// TIA Portal project "MedicalTableS71500" (V15.1)

(* hardware
DEVICE "S71500/ET200MP-Station_1"  S7-1500 station
   slot 0: "Profilschiene_0"  Rack  6ES7 590-1***0-0AA0
   slot 1: "PLC_1"  CPU 1513-1 PN  6ES7 513-1AL02-0AB0  V2.6
      slot 3: "CPU-Display_1"  6ES7591-1AA00-0AA0
   slot 2: "DI 32x24VDC BA_1"  DI 32x24VDC BA  6ES7 521-1BL10-0AA0  V1.0
   slot 3: "AI 8xU/I/RTD/TC ST_1"  AI 8xU/I/RTD/TC ST  6ES7 531-7KF00-0AB0  V2.2
   slot 4: "DQ 32x24VDC/0.5A BA_1"  DQ 32x24VDC/0.5A BA  6ES7 522-1BL10-0AA0  V1.0
   slot 5: "AQ 4xU/I ST_1"  AQ 4xU/I ST  6ES7 532-5HD00-0AB0  V2.2
   slot 6: "DI 16x24VDC BA_1"  DI 16x24VDC BA  6ES7 521-1BH10-0AA0  V1.0
*)

// ===== PLC "PLC_1"  CPU 1513-1 PN =====

VAR_GLOBAL   // PLC tag table "Standard-Variablentabelle"
   "FlagControlOn" AT %M0.0 : Bool;
   "FlagM1ManualPosToMin" AT %M0.1 : Bool;
   "FlagM1ManualPosToMax" AT %M0.2 : Bool;
   "FlagM2ManualPosToMin" AT %M0.3 : Bool;
   "FlagM2ManualPosToMax" AT %M0.4 : Bool;
   "FlagM3ManualPosToMin" AT %M0.5 : Bool;
   "FlagM3ManualPosToMax" AT %M0.6 : Bool;
   "FlagM4ManualPosToMin" AT %M0.7 : Bool;
   "FlagM4ManualPosToMax" AT %M1.0 : Bool;
   "FlagEdgeHelperS5" AT %M1.1 : Bool;
   "FlagEdgeHelperS10" AT %M1.2 : Bool;
   "P2AllPositionsReached" AT %A2.2 : Bool;
   "P3M1PosReached" AT %A2.3 : Bool;
   "P4M2PosReached" AT %A2.4 : Bool;
   "P5M3PosReached" AT %A2.5 : Bool;
   "P6M4PosReached" AT %A2.6 : Bool;
   "FlagNewDataSetHelper" AT %M1.3 : Bool;
   "FlagNewDataSetEdgeHelper" AT %M1.4 : Bool;
   "P7StoreTeachInSettingsDone" AT %A2.7 : Bool;
END_VAR

VAR_GLOBAL   // PLC tag table "Variablentabelle aus XML_1"
   "S1ControlOn" AT %I0.0 : Bool;
   "S2ControlOff" AT %I0.1 : Bool;   // NC
   "S3ModeSetSetting" AT %I0.2 : Bool;   // The current positions are taken over
   "S4ModeTeachIn" AT %I0.3 : Bool;   // The positions can be adjusted manually
   "S5StoreSetting" AT %I0.4 : Bool;   // The saved positions can be selected
   "B1_M1MinPos" AT %I0.5 : Bool;   // NC
   "B2_M1MaxPos" AT %I0.6 : Bool;   // NC
   "B3_M2LeftPos" AT %I0.7 : Bool;   // NC
   "B4_M2RightPos" AT %I1.0 : Bool;   // NC
   "B5_M3MinPos" AT %I1.1 : Bool;   // NC
   "B6_M3MaxPos" AT %I1.2 : Bool;   // NC
   "B7_M4MinPos" AT %I1.3 : Bool;   // NC
   "B8_M4MaxPos" AT %I1.4 : Bool;   // NC
   "S6TeachInGotoMin" AT %I1.5 : Bool;   // Moves the selected drive unit to min. when teach-in mode is selected.
   "S7TeachInGotoMax" AT %I1.6 : Bool;   // Moves the selected drive unit to max. when teach-in mode is selected.
   "S8TeachInSelectedDriveUnit" AT %EB10 : Byte;   // The selected drive unit 1-4
   "B9_M1Position" AT %EW12 : Word;
   "B10_M2Position" AT %EW14 : Int;
   "B11_M3Position" AT %EW16 : Word;
   "B12_M4Position" AT %EW18 : Word;
   "P1ControlOn" AT %Q0.0 : Bool;
   "M1AutomPositioningActive" AT %Q0.1 : Bool;
   "M2AutomPositioningActive" AT %Q0.2 : Bool;
   "M3AutomPositioningActive" AT %Q0.3 : Bool;
   "M4AutomPositioningActive" AT %Q0.4 : Bool;
   "M1ManualPosToMin" AT %Q0.5 : Bool;
   "M1ManualPosToMax" AT %Q0.6 : Bool;
   "M2ManualPosToMin" AT %Q0.7 : Bool;
   "M2ManualPosToMax" AT %Q1.0 : Bool;
   "M3ManualPosToMin" AT %Q1.1 : Bool;
   "M3ManualPosToMax" AT %Q1.2 : Bool;
   "M4ManualPosToMin" AT %Q1.3 : Bool;
   "M4ManualPosToMax" AT %Q1.4 : Bool;
   "P2AutomaticPositioningDone" AT %Q1.5 : Bool;
   "S10SetSettingOfDataSetNo" AT %I2.3 : Bool;   // The selected data set for teach-in or to set the settings
   "S9_DataSetNumber" AT %IB20 : Byte;
   "M1AutomPositioningStart" AT %Q1.6 : Bool;
   "M2AutomPositioningStart" AT %Q1.7 : Bool;
   "M3AutomPositioningStart" AT %Q2.0 : Bool;
   "M4AutomPositioningStart" AT %Q2.1 : Bool;
   "M1TargetPos" AT %QW10 : Word;
   "M2TargetPos" AT %QW12 : Int;
   "M3TargetPos" AT %QW14 : Word;
   "M4TargetPos" AT %QW16 : Word;
   "M1TargetPosReached" AT %I1.7 : Bool;
   "M2TargetPosReached" AT %I2.0 : Bool;
   "M3TargetPosReached" AT %I2.1 : Bool;
   "M4TargetPosReached" AT %I2.2 : Bool;
END_VAR

DATA_BLOCK "DataSettings"   // DB1
{ S7_Optimized_Access := 'TRUE' }
VERSION : 0.1
   VAR
      DataSet : Array[0..3] of Struct
         M1Pos : Int;
         M2Pos : Int;
         M3Pos : Int;
         M4Pos : Int;
      END_STRUCT;
   END_VAR
BEGIN
   DataSet[0].M1Pos := 20;
   DataSet[0].M2Pos := -30;
   DataSet[0].M3Pos := 10;
   DataSet[0].M4Pos := 10;
   DataSet[1].M1Pos := 30;
   DataSet[1].M2Pos := -20;
   DataSet[1].M3Pos := 25;
   DataSet[1].M4Pos := 25;
   DataSet[2].M1Pos := 40;
   DataSet[2].M2Pos := 10;
   DataSet[2].M3Pos := 35;
   DataSet[2].M4Pos := 35;
   DataSet[3].M1Pos := 60;
   DataSet[3].M2Pos := 30;
   DataSet[3].M3Pos := 40;
   DataSet[3].M4Pos := 40;
END_DATA_BLOCK

DATA_BLOCK "SetDataSettingsStepsAndOutputs_DB"   // DB2
{ S7_Optimized_Access := 'TRUE' }
VERSION : 0.1
// stored: InstanceOfName SetDataSettingsStepsAndOutputs
"SetDataSettingsStepsAndOutputs"
BEGIN
END_DATA_BLOCK

FUNCTION_BLOCK "SetDataSettingsStepsAndOutputs"   // FB1, FBD
{ S7_Optimized_Access := 'TRUE' }
VERSION : 0.1
   VAR
      S10EdgeHelper : Bool;
      Step1 : Bool;
      Step2 : Bool;
      Step3 : Bool;
      Step4 : Bool;
      Step5 : Bool;
      Step6 : Bool;
      Step7 : Bool;
      InsideSteps : Bool;
   END_VAR
   VAR_TEMP   // added for the SCL form of the ladder/FBD networks
      _w1 : Bool;
   END_VAR
BEGIN

REGION Network 1: M1 to pos
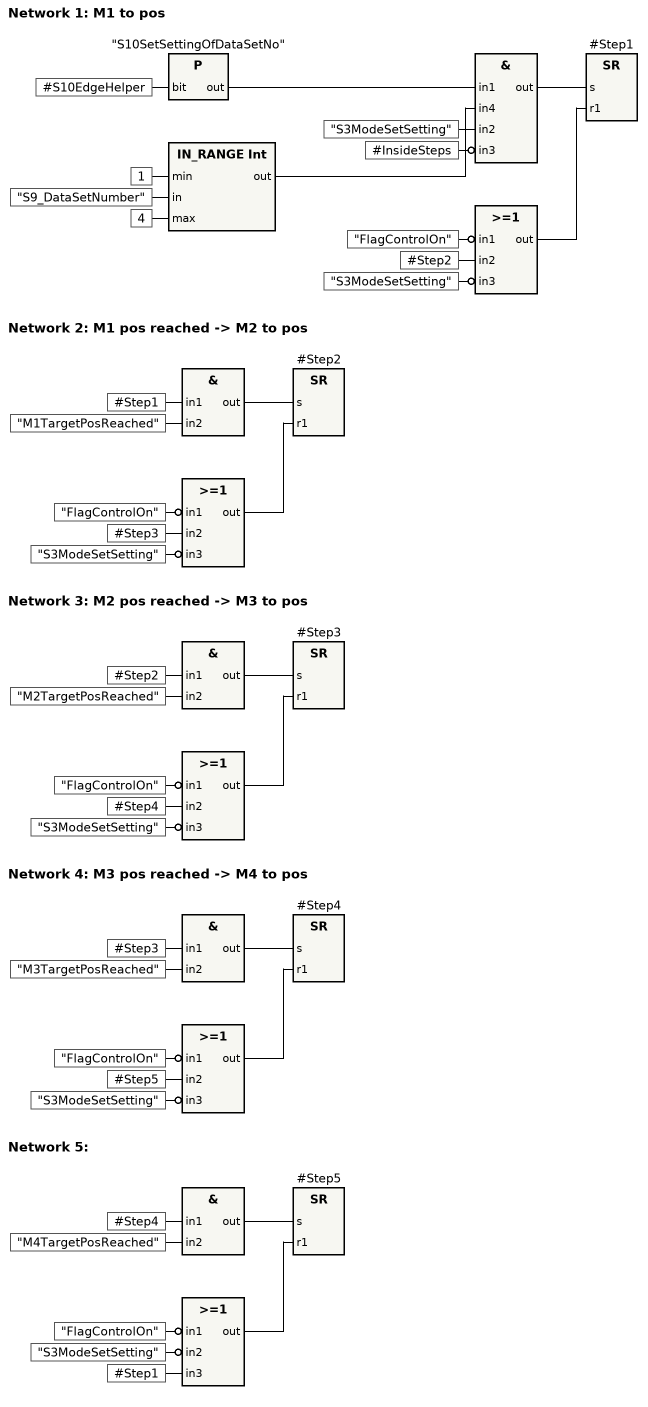
   #_w1 := "S10SetSettingOfDataSetNo" AND NOT #S10EdgeHelper;   // rising edge of "S10SetSettingOfDataSetNo"
   #S10EdgeHelper := "S10SetSettingOfDataSetNo";
   IF #_w1 AND (1 <= "S9_DataSetNumber") AND ("S9_DataSetNumber" <= 4) AND "S3ModeSetSetting" AND NOT #InsideSteps THEN
       #Step1 := TRUE;   // SR flip-flop
   END_IF;
   IF NOT "FlagControlOn" OR #Step2 OR NOT "S3ModeSetSetting" THEN #Step1 := FALSE; END_IF;
END_REGION

REGION Network 2: M1 pos reached -> M2 to pos
   IF #Step1 AND "M1TargetPosReached" THEN
       #Step2 := TRUE;   // SR flip-flop
   END_IF;
   IF NOT "FlagControlOn" OR #Step3 OR NOT "S3ModeSetSetting" THEN #Step2 := FALSE; END_IF;
END_REGION

REGION Network 3: M2 pos reached -> M3 to pos
   IF #Step2 AND "M2TargetPosReached" THEN
       #Step3 := TRUE;   // SR flip-flop
   END_IF;
   IF NOT "FlagControlOn" OR #Step4 OR NOT "S3ModeSetSetting" THEN #Step3 := FALSE; END_IF;
END_REGION

REGION Network 4: M3 pos reached -> M4 to pos
   IF #Step3 AND "M3TargetPosReached" THEN
       #Step4 := TRUE;   // SR flip-flop
   END_IF;
   IF NOT "FlagControlOn" OR #Step5 OR NOT "S3ModeSetSetting" THEN #Step4 := FALSE; END_IF;
END_REGION

REGION Network 5
   IF #Step4 AND "M4TargetPosReached" THEN
       #Step5 := TRUE;   // SR flip-flop
   END_IF;
   IF NOT "FlagControlOn" OR NOT "S3ModeSetSetting" OR #Step1 THEN #Step5 := FALSE; END_IF;
END_REGION

REGION Network 6: Inside steps
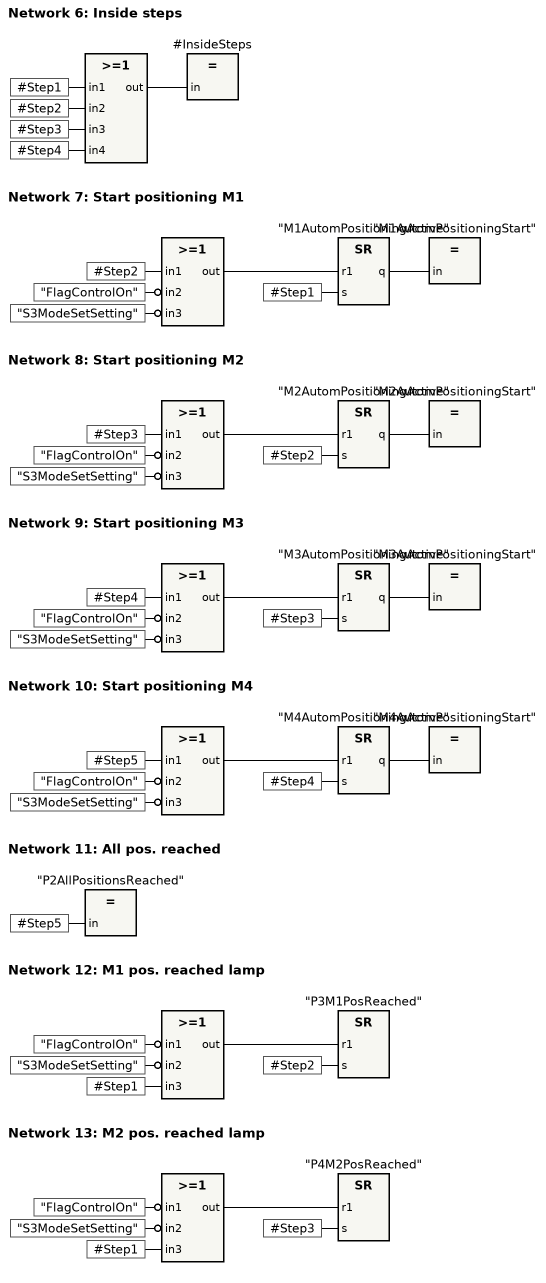
   #InsideSteps := #Step1 OR #Step2 OR #Step3 OR #Step4;
END_REGION

REGION Network 7: Start positioning M1
   IF #Step1 THEN
       "M1AutomPositioningActive" := TRUE;   // SR flip-flop
   END_IF;
   IF #Step2 OR NOT "FlagControlOn" OR NOT "S3ModeSetSetting" THEN
       "M1AutomPositioningActive" := FALSE;
   END_IF;
   "M1AutomPositioningStart" := "M1AutomPositioningActive";
END_REGION

REGION Network 8: Start positioning M2
   IF #Step2 THEN
       "M2AutomPositioningActive" := TRUE;   // SR flip-flop
   END_IF;
   IF #Step3 OR NOT "FlagControlOn" OR NOT "S3ModeSetSetting" THEN
       "M2AutomPositioningActive" := FALSE;
   END_IF;
   "M2AutomPositioningStart" := "M2AutomPositioningActive";
END_REGION

REGION Network 9: Start positioning M3
   IF #Step3 THEN
       "M3AutomPositioningActive" := TRUE;   // SR flip-flop
   END_IF;
   IF #Step4 OR NOT "FlagControlOn" OR NOT "S3ModeSetSetting" THEN
       "M3AutomPositioningActive" := FALSE;
   END_IF;
   "M3AutomPositioningStart" := "M3AutomPositioningActive";
END_REGION

REGION Network 10: Start positioning M4
   IF #Step4 THEN
       "M4AutomPositioningActive" := TRUE;   // SR flip-flop
   END_IF;
   IF #Step5 OR NOT "FlagControlOn" OR NOT "S3ModeSetSetting" THEN
       "M4AutomPositioningActive" := FALSE;
   END_IF;
   "M4AutomPositioningStart" := "M4AutomPositioningActive";
END_REGION

REGION Network 11: All pos. reached
   "P2AllPositionsReached" := #Step5;
END_REGION

REGION Network 12: M1 pos. reached lamp
   IF #Step2 THEN
       "P3M1PosReached" := TRUE;   // SR flip-flop
   END_IF;
   IF NOT "FlagControlOn" OR NOT "S3ModeSetSetting" OR #Step1 THEN "P3M1PosReached" := FALSE; END_IF;
END_REGION

REGION Network 13: M2 pos. reached lamp
   IF #Step3 THEN
       "P4M2PosReached" := TRUE;   // SR flip-flop
   END_IF;
   IF NOT "FlagControlOn" OR NOT "S3ModeSetSetting" OR #Step1 THEN "P4M2PosReached" := FALSE; END_IF;
END_REGION

REGION Network 14: M3 pos. reached lamp
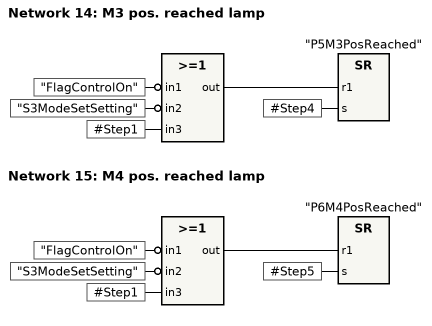
   IF #Step4 THEN
       "P5M3PosReached" := TRUE;   // SR flip-flop
   END_IF;
   IF NOT "FlagControlOn" OR NOT "S3ModeSetSetting" OR #Step1 THEN "P5M3PosReached" := FALSE; END_IF;
END_REGION

REGION Network 15: M4 pos. reached lamp
   IF #Step5 THEN
       "P6M4PosReached" := TRUE;   // SR flip-flop
   END_IF;
   IF NOT "FlagControlOn" OR NOT "S3ModeSetSetting" OR #Step1 THEN "P6M4PosReached" := FALSE; END_IF;
END_REGION
END_FUNCTION_BLOCK

FUNCTION "MHJ-PLC-Lab-Function-S71500" : Void   // FC1, SCL
{ S7_Optimized_Access := 'TRUE' }
VERSION : 0.1
   VAR_INPUT
      MinDiByte : Int;
      MaxDiByte : Int;
   END_VAR
   VAR_TEMP
      Value : Byte;
      ForCounter : Int;
      MaxDiByteTemp : Int;
      MinDiByteTemp : Int;
   END_VAR
   VAR CONSTANT
      Value_01_DW : DWord := 16#1223_5486;
      Value_02_DW : DWord := 16#A6C9_D1F5;
   END_VAR
BEGIN

   #Value:=PEEK(area := 16#82,
        dbNumber := 0,
        byteOffset := 511);
   #Value := #Value + 1;

   POKE(area := 16#82,
        dbNumber := 0,
        byteOffset := 511,
        value := #Value);

   POKE(area := 16#82,
        dbNumber := 0,
        byteOffset := 1016,
        value := #Value_01_DW);
   POKE(area := 16#82,
        dbNumber := 0,
        byteOffset := 1020,
        value := #Value_02_DW);

   #MaxDiByteTemp := 462;
   IF #MaxDiByte < 463 THEN
       #MaxDiByteTemp := #MaxDiByte;
   END_IF;

   #MinDiByteTemp := 0;
   IF #MaxDiByteTemp >= #MinDiByte & #MinDiByte >= 0 THEN
       #MinDiByteTemp := #MinDiByte;
   END_IF;

   FOR #ForCounter := #MinDiByteTemp TO #MaxDiByteTemp DO
       #Value := PEEK(area := 16#1,
                      dbNumber := 0,
                      byteOffset := #ForCounter);
       POKE(area := 16#81,
            dbNumber := 0,
            byteOffset := #ForCounter,
            value := #Value);
   END_FOR;

   #Value := PEEK(area := 16#1,
                  dbNumber := 0,
                  byteOffset := 512);
   POKE(area := 16#82,
        dbNumber := 0,
        byteOffset := 512,
        value := #Value);
END_FUNCTION

FUNCTION "MHJ-PLC-Lab-Function-S71500-NextInputArea" : Void   // FC2, SCL
{ S7_Optimized_Access := 'TRUE' }
VERSION : 0.1
   VAR_INPUT
      MinDiByte : Int;
      MaxDiByte : Int;
   END_VAR
   VAR_TEMP
      Value : Byte;
      ForCounter : Int;
      MaxDiByteTemp : Int;
      MinDiByteTemp : Int;
   END_VAR
BEGIN


   #MaxDiByteTemp := -1;
   IF #MaxDiByte < 463 THEN
       #MaxDiByteTemp := #MaxDiByte;
   END_IF;

   #MinDiByteTemp := -1;
   IF #MaxDiByteTemp >= #MinDiByte & #MinDiByte >= 0 THEN
       #MinDiByteTemp := #MinDiByte;
   END_IF;

   IF #MaxDiByteTemp >= 0 & #MinDiByte >= 0 THEN
       FOR #ForCounter := #MinDiByteTemp TO #MaxDiByteTemp DO
           #Value := PEEK(area := 16#1,
                          dbNumber := 0,
                          byteOffset := #ForCounter);
           POKE(area := 16#81,
                dbNumber := 0,
                byteOffset := #ForCounter,
                value := #Value);
       END_FOR;

   END_IF;
END_FUNCTION

FUNCTION "TeachInDriveUnits" : Void   // FC3, FBD
{ S7_Optimized_Access := 'TRUE' }
VERSION : 0.1
BEGIN

REGION Network 1
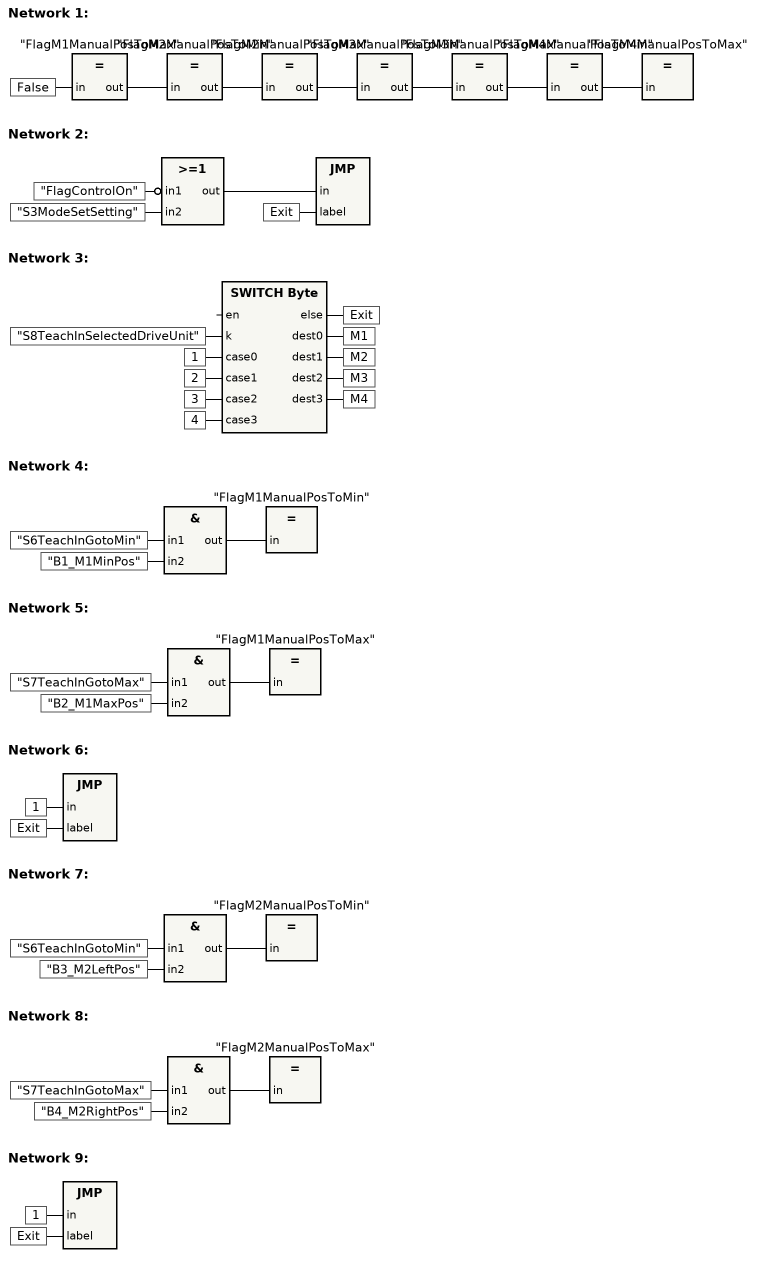
   "FlagM1ManualPosToMax" := False;
   "FlagM2ManualPosToMin" := False;
   "FlagM2ManualPosToMax" := False;
   "FlagM3ManualPosToMin" := False;
   "FlagM3ManualPosToMax" := False;
   "FlagM4ManualPosToMin" := False;
   "FlagM4ManualPosToMax" := False;
END_REGION

REGION Network 2
   IF NOT "FlagControlOn" OR "S3ModeSetSetting" THEN GOTO Exit; END_IF;
END_REGION

REGION Network 3
   // no SCL statement known for Switch: written as a call
   Switch(k := "S8TeachInSelectedDriveUnit",
          case0 := 1,
          case1 := 2,
          case2 := 3,
          case3 := 4,
          "else" => Exit,
          dest0 => M1,
          dest1 => M2,
          dest2 => M3,
          dest3 => M4);
END_REGION

REGION Network 4
   M1:
   "FlagM1ManualPosToMin" := "S6TeachInGotoMin" AND "B1_M1MinPos";
END_REGION

REGION Network 5
   "FlagM1ManualPosToMax" := "S7TeachInGotoMax" AND "B2_M1MaxPos";
END_REGION

REGION Network 6
   IF 1 THEN GOTO Exit; END_IF;
END_REGION

REGION Network 7
   M2:
   "FlagM2ManualPosToMin" := "S6TeachInGotoMin" AND "B3_M2LeftPos";
END_REGION

REGION Network 8
   "FlagM2ManualPosToMax" := "S7TeachInGotoMax" AND "B4_M2RightPos";
END_REGION

REGION Network 9
   IF 1 THEN GOTO Exit; END_IF;
END_REGION

REGION Network 10
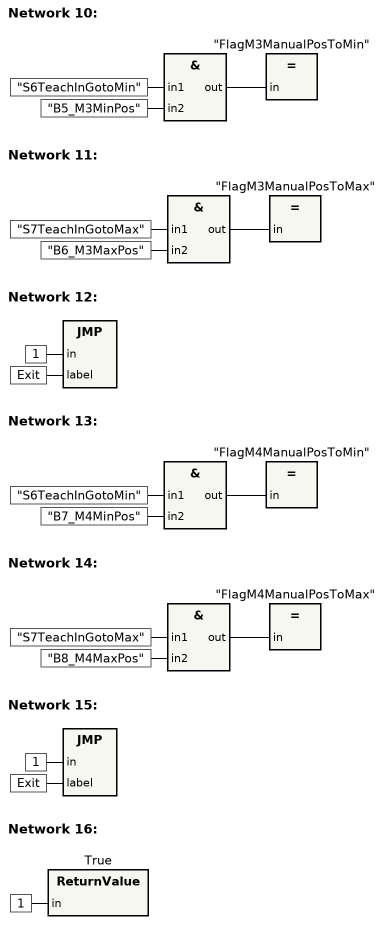
   M3:
   "FlagM3ManualPosToMin" := "S6TeachInGotoMin" AND "B5_M3MinPos";
END_REGION

REGION Network 11
   "FlagM3ManualPosToMax" := "S7TeachInGotoMax" AND "B6_M3MaxPos";
END_REGION

REGION Network 12
   IF 1 THEN GOTO Exit; END_IF;
END_REGION

REGION Network 13
   M4:
   "FlagM4ManualPosToMin" := "S6TeachInGotoMin" AND "B7_M4MinPos";
END_REGION

REGION Network 14
   "FlagM4ManualPosToMax" := "S7TeachInGotoMax" AND "B8_M4MaxPos";
END_REGION

REGION Network 15
   IF 1 THEN GOTO Exit; END_IF;
END_REGION

REGION Network 16
   Exit:
   IF 1 THEN
       ENO := True;
       RETURN;
   END_IF;
END_REGION
END_FUNCTION

FUNCTION "StoreTeachInDataSettings" : Void   // FC4, FBD
{ S7_Optimized_Access := 'TRUE' }
VERSION : 0.1
   VAR_TEMP   // added for the SCL form of the ladder/FBD networks
      _w1 : Bool;
   END_VAR
BEGIN

REGION Network 1
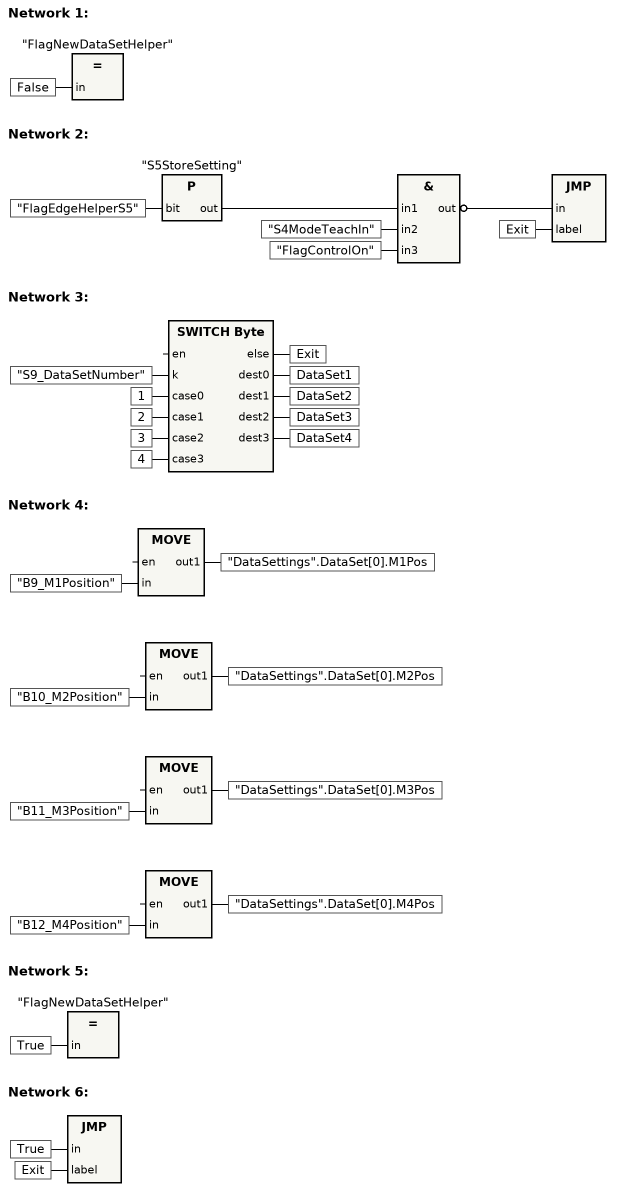
   "FlagNewDataSetHelper" := False;
END_REGION

REGION Network 2
   #_w1 := "S5StoreSetting" AND NOT "FlagEdgeHelperS5";   // rising edge of "S5StoreSetting"
   "FlagEdgeHelperS5" := "S5StoreSetting";
   IF NOT (#_w1 AND "S4ModeTeachIn" AND "FlagControlOn") THEN GOTO Exit; END_IF;
END_REGION

REGION Network 3
   // no SCL statement known for Switch: written as a call
   Switch(k := "S9_DataSetNumber",
          case0 := 1,
          case1 := 2,
          case2 := 3,
          case3 := 4,
          "else" => Exit,
          dest0 => DataSet1,
          dest1 => DataSet2,
          dest2 => DataSet3,
          dest3 => DataSet4);
END_REGION

REGION Network 4
   DataSet1:
   "DataSettings".DataSet[0].M1Pos := "B9_M1Position";
   "DataSettings".DataSet[0].M2Pos := "B10_M2Position";
   "DataSettings".DataSet[0].M3Pos := "B11_M3Position";
   "DataSettings".DataSet[0].M4Pos := "B12_M4Position";
END_REGION

REGION Network 5
   "FlagNewDataSetHelper" := True;
END_REGION

REGION Network 6
   IF True THEN GOTO Exit; END_IF;
END_REGION

REGION Network 7
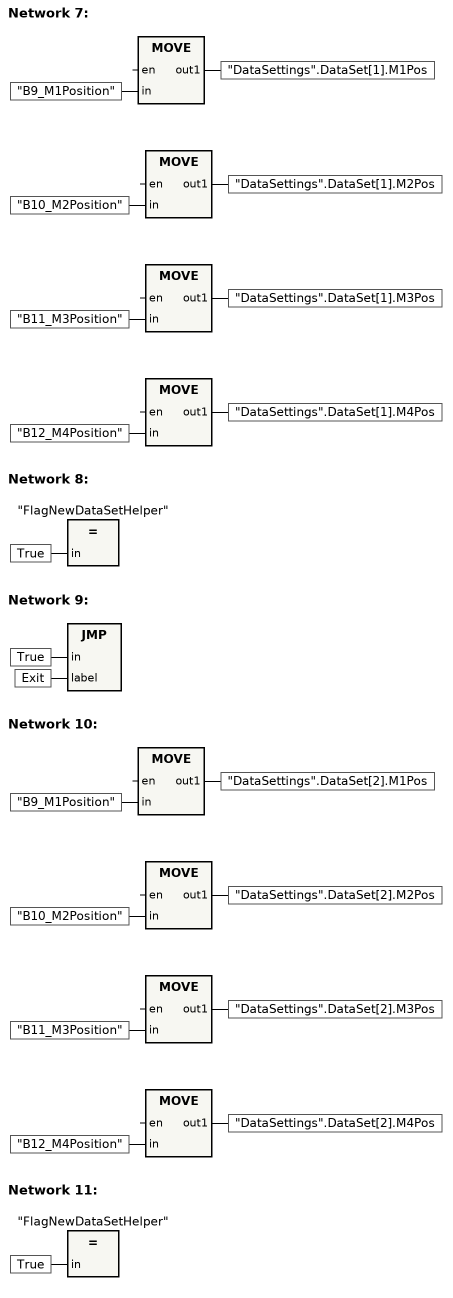
   DataSet2:
   "DataSettings".DataSet[1].M1Pos := "B9_M1Position";
   "DataSettings".DataSet[1].M2Pos := "B10_M2Position";
   "DataSettings".DataSet[1].M3Pos := "B11_M3Position";
   "DataSettings".DataSet[1].M4Pos := "B12_M4Position";
END_REGION

REGION Network 8
   "FlagNewDataSetHelper" := True;
END_REGION

REGION Network 9
   IF True THEN GOTO Exit; END_IF;
END_REGION

REGION Network 10
   DataSet3:
   "DataSettings".DataSet[2].M1Pos := "B9_M1Position";
   "DataSettings".DataSet[2].M2Pos := "B10_M2Position";
   "DataSettings".DataSet[2].M3Pos := "B11_M3Position";
   "DataSettings".DataSet[2].M4Pos := "B12_M4Position";
END_REGION

REGION Network 11
   "FlagNewDataSetHelper" := True;
END_REGION

REGION Network 12
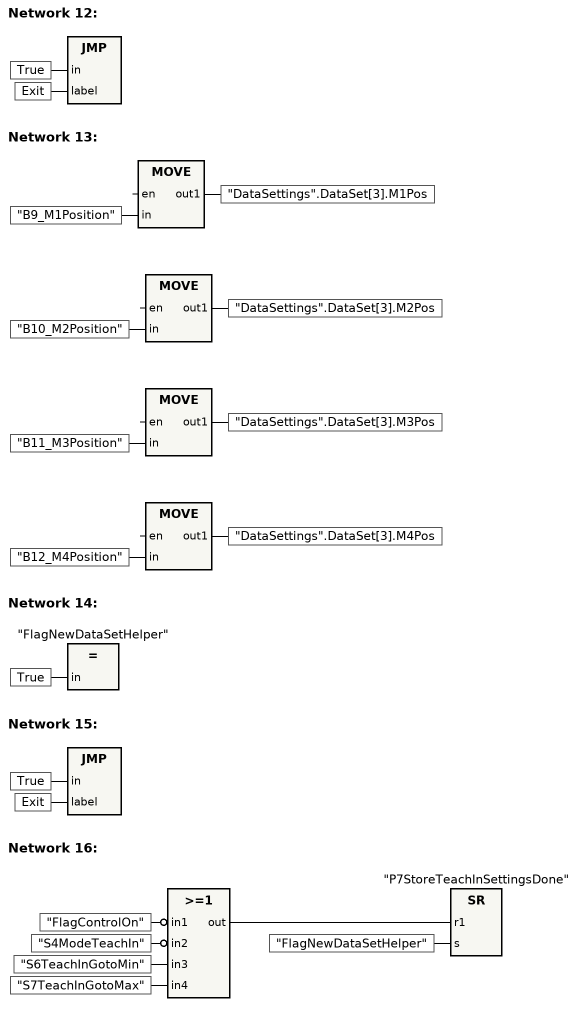
   IF True THEN GOTO Exit; END_IF;
END_REGION

REGION Network 13
   DataSet4:
   "DataSettings".DataSet[3].M1Pos := "B9_M1Position";
   "DataSettings".DataSet[3].M2Pos := "B10_M2Position";
   "DataSettings".DataSet[3].M3Pos := "B11_M3Position";
   "DataSettings".DataSet[3].M4Pos := "B12_M4Position";
END_REGION

REGION Network 14
   "FlagNewDataSetHelper" := True;
END_REGION

REGION Network 15
   IF True THEN GOTO Exit; END_IF;
END_REGION

REGION Network 16
   Exit:
   IF "FlagNewDataSetHelper" THEN
       "P7StoreTeachInSettingsDone" := TRUE;   // SR flip-flop
   END_IF;
   IF NOT "FlagControlOn" OR NOT "S4ModeTeachIn" OR "S6TeachInGotoMin" OR "S7TeachInGotoMax" THEN
       "P7StoreTeachInSettingsDone" := FALSE;
   END_IF;
END_REGION
END_FUNCTION

FUNCTION "SetDataSettingsData" : Void   // FC5, FBD
{ S7_Optimized_Access := 'TRUE' }
VERSION : 0.1
   VAR_TEMP   // added for the SCL form of the ladder/FBD networks
      _w1 : Bool;
   END_VAR
BEGIN

REGION Network 1
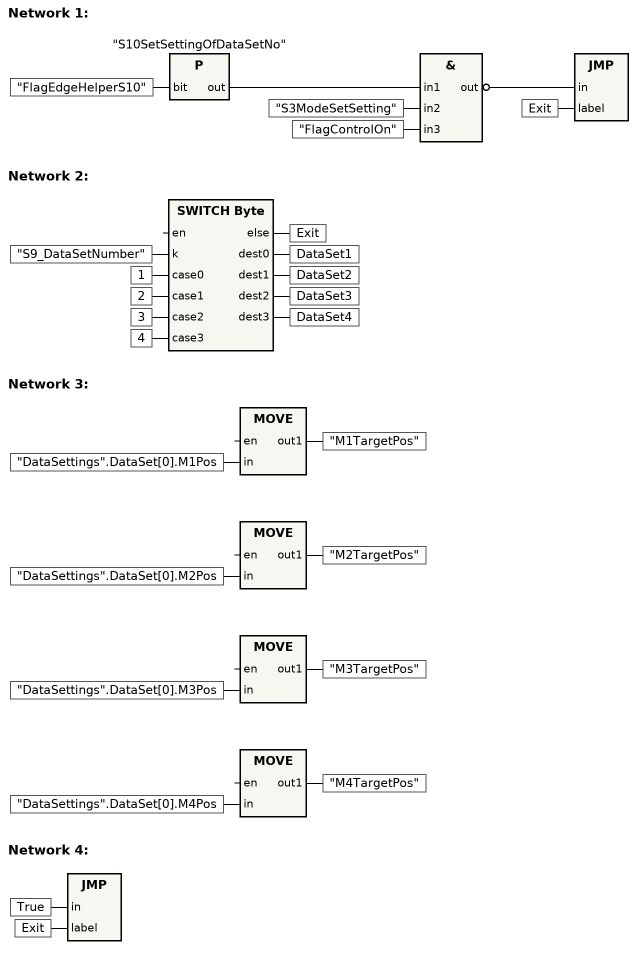
   #_w1 := "S10SetSettingOfDataSetNo" AND NOT "FlagEdgeHelperS10";   // rising edge of "S10SetSettingOfDataSetNo"
   "FlagEdgeHelperS10" := "S10SetSettingOfDataSetNo";
   IF NOT (#_w1 AND "S3ModeSetSetting" AND "FlagControlOn") THEN GOTO Exit; END_IF;
END_REGION

REGION Network 2
   // no SCL statement known for Switch: written as a call
   Switch(k := "S9_DataSetNumber",
          case0 := 1,
          case1 := 2,
          case2 := 3,
          case3 := 4,
          "else" => Exit,
          dest0 => DataSet1,
          dest1 => DataSet2,
          dest2 => DataSet3,
          dest3 => DataSet4);
END_REGION

REGION Network 3
   DataSet1:
   "M1TargetPos" := "DataSettings".DataSet[0].M1Pos;
   "M2TargetPos" := "DataSettings".DataSet[0].M2Pos;
   "M3TargetPos" := "DataSettings".DataSet[0].M3Pos;
   "M4TargetPos" := "DataSettings".DataSet[0].M4Pos;
END_REGION

REGION Network 4
   IF True THEN GOTO Exit; END_IF;
END_REGION

REGION Network 5
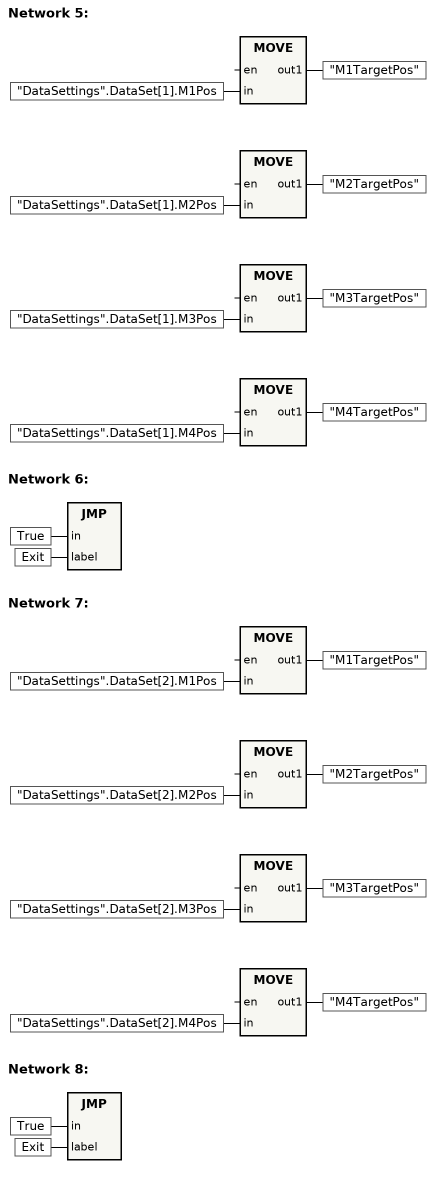
   DataSet2:
   "M1TargetPos" := "DataSettings".DataSet[1].M1Pos;
   "M2TargetPos" := "DataSettings".DataSet[1].M2Pos;
   "M3TargetPos" := "DataSettings".DataSet[1].M3Pos;
   "M4TargetPos" := "DataSettings".DataSet[1].M4Pos;
END_REGION

REGION Network 6
   IF True THEN GOTO Exit; END_IF;
END_REGION

REGION Network 7
   DataSet3:
   "M1TargetPos" := "DataSettings".DataSet[2].M1Pos;
   "M2TargetPos" := "DataSettings".DataSet[2].M2Pos;
   "M3TargetPos" := "DataSettings".DataSet[2].M3Pos;
   "M4TargetPos" := "DataSettings".DataSet[2].M4Pos;
END_REGION

REGION Network 8
   IF True THEN GOTO Exit; END_IF;
END_REGION

REGION Network 9
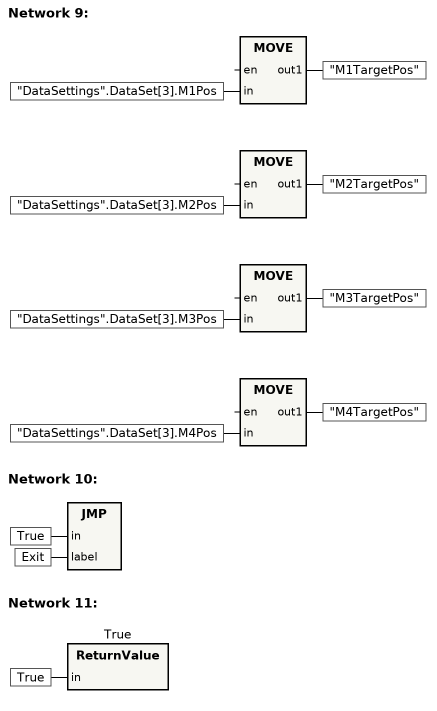
   DataSet4:
   "M1TargetPos" := "DataSettings".DataSet[3].M1Pos;
   "M2TargetPos" := "DataSettings".DataSet[3].M2Pos;
   "M3TargetPos" := "DataSettings".DataSet[3].M3Pos;
   "M4TargetPos" := "DataSettings".DataSet[3].M4Pos;
END_REGION

REGION Network 10
   IF True THEN GOTO Exit; END_IF;
END_REGION

REGION Network 11
   Exit:
   IF True THEN
       ENO := True;
       RETURN;
   END_IF;
END_REGION
END_FUNCTION

FUNCTION "SetTeachInOutputs" : Void   // FC6, FBD
{ S7_Optimized_Access := 'TRUE' }
VERSION : 0.1
BEGIN

REGION Network 1: M1 to max
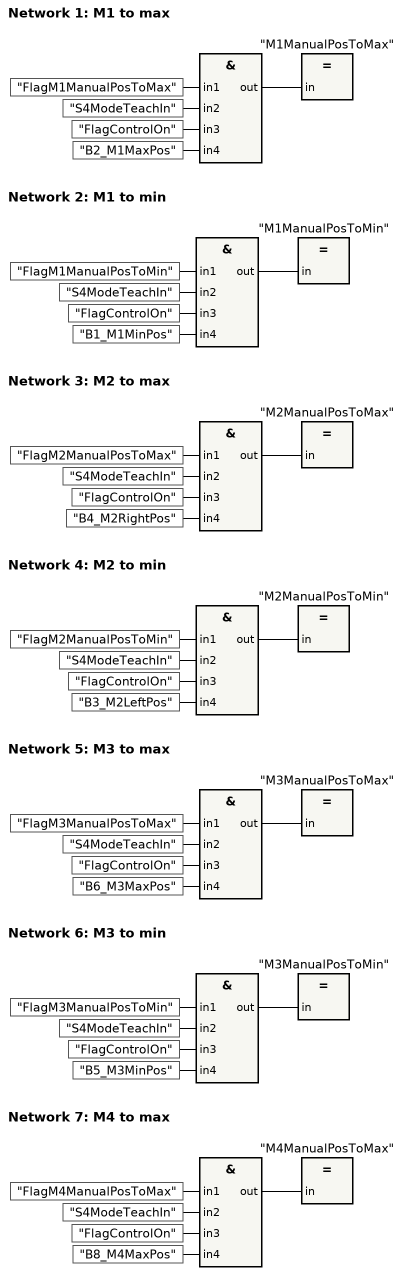
   "M1ManualPosToMax" := "FlagM1ManualPosToMax" AND "S4ModeTeachIn" AND "FlagControlOn" AND "B2_M1MaxPos";
END_REGION

REGION Network 2: M1 to min
   "M1ManualPosToMin" := "FlagM1ManualPosToMin" AND "S4ModeTeachIn" AND "FlagControlOn" AND "B1_M1MinPos";
END_REGION

REGION Network 3: M2 to max
   "M2ManualPosToMax" := "FlagM2ManualPosToMax" AND "S4ModeTeachIn" AND "FlagControlOn" AND "B4_M2RightPos";
END_REGION

REGION Network 4: M2 to min
   "M2ManualPosToMin" := "FlagM2ManualPosToMin" AND "S4ModeTeachIn" AND "FlagControlOn" AND "B3_M2LeftPos";
END_REGION

REGION Network 5: M3 to max
   "M3ManualPosToMax" := "FlagM3ManualPosToMax" AND "S4ModeTeachIn" AND "FlagControlOn" AND "B6_M3MaxPos";
END_REGION

REGION Network 6: M3 to min
   "M3ManualPosToMin" := "FlagM3ManualPosToMin" AND "S4ModeTeachIn" AND "FlagControlOn" AND "B5_M3MinPos";
END_REGION

REGION Network 7: M4 to max
   "M4ManualPosToMax" := "FlagM4ManualPosToMax" AND "S4ModeTeachIn" AND "FlagControlOn" AND "B8_M4MaxPos";
END_REGION

REGION Network 8: M4 to min
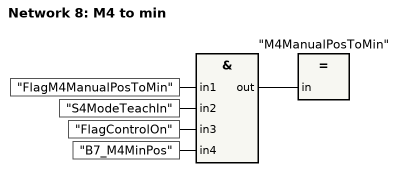
   "M4ManualPosToMin" := "FlagM4ManualPosToMin" AND "S4ModeTeachIn" AND "FlagControlOn" AND "B7_M4MinPos";
END_REGION
END_FUNCTION

ORGANIZATION_BLOCK "Main"   // OB1, FBD, ProgramCycle
TITLE = "Main Program Sweep (Cycle)"
{ S7_Optimized_Access := 'TRUE' }
VERSION : 0.1
   VAR_INPUT
      Initial_Call : Bool;   // Initial call of this OB
      Remanence : Bool;   // =True, if remanent data are available
   END_VAR
   VAR_TEMP   // added for the SCL form of the ladder/FBD networks
      _w1 : Bool;
   END_VAR
BEGIN

REGION Network 1
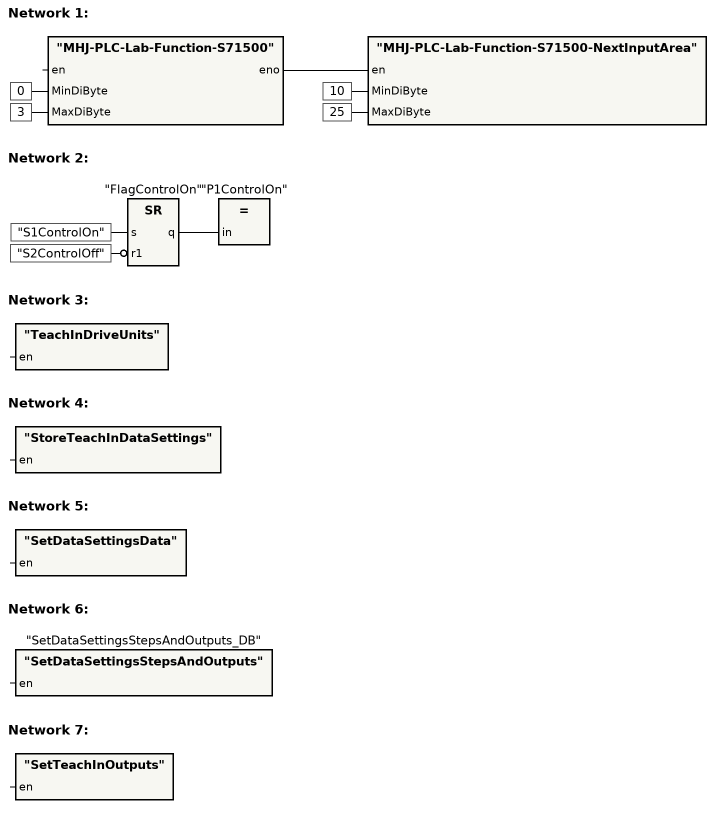
   "MHJ-PLC-Lab-Function-S71500"(MinDiByte := 0, MaxDiByte := 3, ENO => #_w1);
   IF #_w1 THEN "MHJ-PLC-Lab-Function-S71500-NextInputArea"(MinDiByte := 10, MaxDiByte := 25); END_IF;
END_REGION

REGION Network 2
   IF "S1ControlOn" THEN
       "FlagControlOn" := TRUE;   // SR flip-flop
   END_IF;
   IF NOT "S2ControlOff" THEN "FlagControlOn" := FALSE; END_IF;
   "P1ControlOn" := "FlagControlOn";
END_REGION

REGION Network 3
   "TeachInDriveUnits"();
END_REGION

REGION Network 4
   "StoreTeachInDataSettings"();
END_REGION

REGION Network 5
   "SetDataSettingsData"();
END_REGION

REGION Network 6
   "SetDataSettingsStepsAndOutputs_DB"();   // "SetDataSettingsStepsAndOutputs"
END_REGION

REGION Network 7
   "SetTeachInOutputs"();
END_REGION
END_ORGANIZATION_BLOCK